# B&R Automation Studio project AS_Target_Simulink_Test (part 5)

#### TD_Test.c
```c
/********************************************************************
 * COPYRIGHT -- Bernecker + Rainer Industrie-Elektronik Ges.m.b.H.
 ********************************************************************
 * Program: TransmissionDownshiftTestSequence
 * File: TD_Test.c
 * Author: The MathWorks, Inc.
 * Created: Wed Jun 03 01:12:01 1998
 ********************************************************************
 * Implementation of program TransmissionDownshiftTestSequence
 ********************************************************************
 * Generated with B&R Automation Studio Target for Simulink  V6.1.0
 * (ERT based)
 ********************************************************************/

#define _ASMATH_
#define ASMATH_
#define _ASMATH_H
#define ASMATH_H
#define _ASMATH_H_
#define ASMATH_H_
#define _ASSTRING_
#define ASSTRING_
#define _ASSTRING_H
#define ASSTRING_H
#define _ASSTRING_H_
#define ASSTRING_H_
#include <bur/plctypes.h>
#ifdef _DEFAULT_INCLUDES
#include <AsDefault.h>
#endif

#include "TransmissionDownshiftTestSequence.h"
#include "rtwtypes.h"

/*  Defines */

/*  Data Types */

/**************************** GLOBAL DATA *************************************/
/*  Definitions */

/*  Declarations  */

/***************************** FILE SCOPE DATA ********************************/

/*************************** FUNCTIONS ****************************************/
#ifdef __cplusplus

unsigned long bur_heap_size = 6553500;

#endif

  void _INIT mainINIT(void)
{

    UDINT st_ident;
  RTInfo_typ rt_info;
  rt_info.enable = 1;
  RTInfo(&rt_info);
  if (rt_info.cycle_time != 10000) {
    /* cycle time does not match Simulink fixed-step size */
    ST_ident("TD_Test", 0, &st_ident);
    ST_tmp_suspend(st_ident);
    ERR_warning(33310, 0);
  }

  /* initialize model */
  TransmissionDownshiftTestSequence_initialize();

} void _CYCLIC mainCYCLIC(void)
{
  /* call model step function */
  TransmissionDownshiftTestSequence_output();

  TransmissionDownshiftTestSequence_update();

} void _EXIT mainEXIT(void)
{
  /* terminate model */
  TransmissionDownshiftTestSequence_terminate();

} /*****************************************************************************
     Task sample time: 0.01s
   *****************************************************************************/
/*****************************************************************************
   B&R Automation Studio Target for Simulink Version: V6.1.0 (06-Nov-2019)
 *****************************************************************************/

/*======================== TOOL VERSION INFORMATION ==========================*
 * MATLAB 9.7 (R2019b)18-Jul-2019                                             *
 * Simulink 10.0 (R2019b)18-Jul-2019                                          *
 * Simulink Coder 9.2 (R2019b)18-Jul-2019                                     *
 * Embedded Coder 7.3 (R2019b)18-Jul-2019                                     *
 * Stateflow 10.1 (R2019b)18-Jul-2019                                         *
 * Fixed-Point Designer 6.4 (R2019b)18-Jul-2019                               *
 *============================================================================*/

/*======================= LICENSE IN USE INFORMATION =========================*
 * matlab                                                                     *
 * matlab_coder                                                               *
 * real-time_workshop                                                         *
 * rtw_embedded_coder                                                         *
 * simulink                                                                   *
 * simulink_test                                                              *
 * stateflow                                                                  *
 *============================================================================*/
```

#### TransmissionDownshiftTestSequence.c
```c
/********************************************************************
 * COPYRIGHT -- Bernecker + Rainer Industrie-Elektronik Ges.m.b.H.
 ********************************************************************
 * Program: TransmissionDownshiftTestSequence
 * File: TransmissionDownshiftTestSequence.c
 * Author: The MathWorks, Inc.
 * Created: Wed Jun 03 01:12:01 1998
 ********************************************************************
 * Implementation of program TransmissionDownshiftTestSequence
 ********************************************************************
 * Generated with B&R Automation Studio Target for Simulink  V6.1.0
 * (ERT based)
 ********************************************************************/

#include "TransmissionDownshiftTestSequence.h"
#include "TransmissionDownshiftTestSequence_private.h"

/*  Defines */

/* Named constants for Chart: '<Root>/shift_controller' */
#define TransmissionDow_IN_downshifting ((uint8_T)1U)
#define TransmissionDow_IN_steady_state ((uint8_T)2U)
#define TransmissionDowns_IN_upshifting ((uint8_T)3U)
#define TransmissionDownshif_event_DOWN (0)
#define TransmissionDownshiftT_event_UP (1)
#define Transmission_IN_NO_ACTIVE_CHILD ((uint8_T)0U)

/*  Data Types */

/**************************** GLOBAL DATA *************************************/
/*  Definitions */

/* Block signals (default storage) */
BlockIO_TransmissionDownshiftTe TransmissionDownshiftTestSequ_B;

/* Continuous states */
ContinuousStates_TransmissionDo TransmissionDownshiftTestSequ_X;

/* Block states (default storage) */
D_Work_TransmissionDownshiftTes TransmissionDownshiftTest_DWork;

/* External inputs (root inport signals with default storage) */
ExternalInputs_TransmissionDown TransmissionDownshiftTestSequ_U;

/* External outputs (root outports fed by signals with default storage) */
ExternalOutputs_TransmissionDow TransmissionDownshiftTestSequ_Y;

/* Real-time model */
RT_MODEL_TransmissionDownshiftT TransmissionDownshiftTestSeq_M_;
RT_MODEL_TransmissionDownshiftT *const TransmissionDownshiftTestSeq_M =
  &TransmissionDownshiftTestSeq_M_;

/*  Declarations  */

/* Forward declaration for local functions */
static void TransmissionDownshif_gear_state(const int32_T *sfEvent);
static void rate_scheduler(void);

/***************************** FILE SCOPE DATA ********************************/

/*************************** FUNCTIONS ****************************************/
real_T look1_binlxpw(real_T u0, const real_T bp0[], const real_T table[],
                     uint32_T maxIndex)
{
  real_T frac;
  uint32_T iRght;
  uint32_T iLeft;
  uint32_T bpIdx;

  /* Column-major Lookup 1-D
     Search method: 'binary'
     Use previous index: 'off'
     Interpolation method: 'Linear point-slope'
     Extrapolation method: 'Linear'
     Use last breakpoint for index at or above upper limit: 'off'
     Remove protection against out-of-range input in generated code: 'off'
   */
  /* Prelookup - Index and Fraction
     Index Search method: 'binary'
     Extrapolation method: 'Linear'
     Use previous index: 'off'
     Use last breakpoint for index at or above upper limit: 'off'
     Remove protection against out-of-range input in generated code: 'off'
   */
  if (u0 <= bp0[0U]) {
    iLeft = 0U;
    frac = (u0 - bp0[0U]) / (bp0[1U] - bp0[0U]);
  } else if (u0 < bp0[maxIndex]) {
    /* Binary Search */
    bpIdx = maxIndex >> 1U;
    iLeft = 0U;
    iRght = maxIndex;
    while (iRght - iLeft > 1U) {
      if (u0 < bp0[bpIdx]) {
        iRght = bpIdx;
      } else {
        iLeft = bpIdx;
      }

      bpIdx = (iRght + iLeft) >> 1U;
    }

    frac = (u0 - bp0[iLeft]) / (bp0[iLeft + 1U] - bp0[iLeft]);
  } else {
    iLeft = maxIndex - 1U;
    frac = (u0 - bp0[maxIndex - 1U]) / (bp0[maxIndex] - bp0[maxIndex - 1U]);
  }

  /* Column-major Interpolation 1-D
     Interpolation method: 'Linear point-slope'
     Use last breakpoint for index at or above upper limit: 'off'
     Overflow mode: 'portable wrapping'
   */
  return (table[iLeft + 1U] - table[iLeft]) * frac + table[iLeft];
}

real_T look2_binlxpw(real_T u0, real_T u1, const real_T bp0[], const real_T bp1[],
                     const real_T table[], const uint32_T maxIndex[], uint32_T
                     stride)
{
  real_T frac;
  uint32_T bpIndices[2];
  real_T fractions[2];
  real_T yL_1d;
  uint32_T iRght;
  uint32_T bpIdx;
  uint32_T iLeft;

  /* Column-major Lookup 2-D
     Search method: 'binary'
     Use previous index: 'off'
     Interpolation method: 'Linear point-slope'
     Extrapolation method: 'Linear'
     Use last breakpoint for index at or above upper limit: 'off'
     Remove protection against out-of-range input in generated code: 'off'
   */
  /* Prelookup - Index and Fraction
     Index Search method: 'binary'
     Extrapolation method: 'Linear'
     Use previous index: 'off'
     Use last breakpoint for index at or above upper limit: 'off'
     Remove protection against out-of-range input in generated code: 'off'
   */
  if (u0 <= bp0[0U]) {
    iLeft = 0U;
    frac = (u0 - bp0[0U]) / (bp0[1U] - bp0[0U]);
  } else if (u0 < bp0[maxIndex[0U]]) {
    /* Binary Search */
    bpIdx = maxIndex[0U] >> 1U;
    iLeft = 0U;
    iRght = maxIndex[0U];
    while (iRght - iLeft > 1U) {
      if (u0 < bp0[bpIdx]) {
        iRght = bpIdx;
      } else {
        iLeft = bpIdx;
      }

      bpIdx = (iRght + iLeft) >> 1U;
    }

    frac = (u0 - bp0[iLeft]) / (bp0[iLeft + 1U] - bp0[iLeft]);
  } else {
    iLeft = maxIndex[0U] - 1U;
    frac = (u0 - bp0[maxIndex[0U] - 1U]) / (bp0[maxIndex[0U]] - bp0[maxIndex[0U]
      - 1U]);
  }

  fractions[0U] = frac;
  bpIndices[0U] = iLeft;

  /* Prelookup - Index and Fraction
     Index Search method: 'binary'
     Extrapolation method: 'Linear'
     Use previous index: 'off'
     Use last breakpoint for index at or above upper limit: 'off'
     Remove protection against out-of-range input in generated code: 'off'
   */
  if (u1 <= bp1[0U]) {
    iLeft = 0U;
    frac = (u1 - bp1[0U]) / (bp1[1U] - bp1[0U]);
  } else if (u1 < bp1[maxIndex[1U]]) {
    /* Binary Search */
    bpIdx = maxIndex[1U] >> 1U;
    iLeft = 0U;
    iRght = maxIndex[1U];
    while (iRght - iLeft > 1U) {
      if (u1 < bp1[bpIdx]) {
        iRght = bpIdx;
      } else {
        iLeft = bpIdx;
      }

      bpIdx = (iRght + iLeft) >> 1U;
    }

    frac = (u1 - bp1[iLeft]) / (bp1[iLeft + 1U] - bp1[iLeft]);
  } else {
    iLeft = maxIndex[1U] - 1U;
    frac = (u1 - bp1[maxIndex[1U] - 1U]) / (bp1[maxIndex[1U]] - bp1[maxIndex[1U]
      - 1U]);
  }

  /* Column-major Interpolation 2-D
     Interpolation method: 'Linear point-slope'
     Use last breakpoint for index at or above upper limit: 'off'
     Overflow mode: 'portable wrapping'
   */
  bpIdx = iLeft * stride + bpIndices[0U];
  yL_1d = (table[bpIdx + 1U] - table[bpIdx]) * fractions[0U] + table[bpIdx];
  bpIdx += stride;
  return (((table[bpIdx + 1U] - table[bpIdx]) * fractions[0U] + table[bpIdx]) -
          yL_1d) * frac + yL_1d;
}

/*
 *   This function updates active task flag for each subrate.
 * The function is called at model base rate, hence the
 * generated code self-manages all its subrates.
 */
static void rate_scheduler(void)
{
  /* Compute which subrates run during the next base time step.  Subrates
   * are an integer multiple of the base rate counter.  Therefore, the subtask
   * counter is reset when it reaches its limit (zero means run).
   */
  (TransmissionDownshiftTestSeq_M->Timing.TaskCounters.TID[2])++;
  if ((TransmissionDownshiftTestSeq_M->Timing.TaskCounters.TID[2]) > 3) {/* Sample time: [0.04s, 0.0s] */
    TransmissionDownshiftTestSeq_M->Timing.TaskCounters.TID[2] = 0;
  }
}

/*
 * This function updates continuous states using the ODE1 fixed-step
 * solver algorithm
 */
static void rt_ertODEUpdateContinuousStates(RTWSolverInfo *si )
{
  time_T tnew = rtsiGetSolverStopTime(si);
  time_T h = rtsiGetStepSize(si);
  real_T *x = rtsiGetContStates(si);
  ODE1_IntgData *id = (ODE1_IntgData *)rtsiGetSolverData(si);
  real_T *f0 = id->f[0];
  int_T i;
  int_T nXc = 2;
  rtsiSetSimTimeStep(si,MINOR_TIME_STEP);
  rtsiSetdX(si, f0);
  TransmissionDownshiftTestSequence_derivatives();
  rtsiSetT(si, tnew);
  for (i = 0; i < nXc; ++i) {
    x[i] += h * f0[i];
  }

  rtsiSetSimTimeStep(si,MAJOR_TIME_STEP);
}

/* Function for Chart: '<Root>/shift_controller' */
static void TransmissionDownshif_gear_state(const int32_T *sfEvent)
{
  switch (TransmissionDownshiftTestSequ_B.gear) {
   case gearType_first:
    if (*sfEvent == TransmissionDownshiftT_event_UP) {
      TransmissionDownshiftTestSequ_B.gear = gearType_second;
    }
    break;

   case gearType_second:
    if (*sfEvent == TransmissionDownshiftT_event_UP) {
      TransmissionDownshiftTestSequ_B.gear = gearType_third;
    } else {
      if (*sfEvent == TransmissionDownshif_event_DOWN) {
        TransmissionDownshiftTestSequ_B.gear = gearType_first;
      }
    }
    break;

   case gearType_third:
    if (*sfEvent == TransmissionDownshiftT_event_UP) {
      TransmissionDownshiftTestSequ_B.gear = gearType_fourth;
    } else {
      if (*sfEvent == TransmissionDownshif_event_DOWN) {
        TransmissionDownshiftTestSequ_B.gear = gearType_second;
      }
    }
    break;

   case gearType_fourth:
    if (*sfEvent == TransmissionDownshif_event_DOWN) {
      TransmissionDownshiftTestSequ_B.gear = gearType_third;
    }
    break;

   default:
    /* Unreachable state, for coverage only */
    TransmissionDownshiftTestSequ_B.gear = gearType_None;
    break;
  }
}

/* Model output function */
void TransmissionDownshiftTestSequence_output(void)
{
  real_T rtb_out;
  real_T mph;
  int32_T sfEvent;
  real_T interp_down;
  real_T mph_0;
  if (rtmIsMajorTimeStep(TransmissionDownshiftTestSeq_M)) {
    /* set solver stop time */
    if (!(TransmissionDownshiftTestSeq_M->Timing.clockTick0+1)) {
      rtsiSetSolverStopTime(&TransmissionDownshiftTestSeq_M->solverInfo,
                            ((TransmissionDownshiftTestSeq_M->Timing.clockTickH0
        + 1) * TransmissionDownshiftTestSeq_M->Timing.stepSize0 * 4294967296.0));
    } else {
      rtsiSetSolverStopTime(&TransmissionDownshiftTestSeq_M->solverInfo,
                            ((TransmissionDownshiftTestSeq_M->Timing.clockTick0
        + 1) * TransmissionDownshiftTestSeq_M->Timing.stepSize0 +
        TransmissionDownshiftTestSeq_M->Timing.clockTickH0 *
        TransmissionDownshiftTestSeq_M->Timing.stepSize0 * 4294967296.0));
    }
  }                                    /* end MajorTimeStep */

  /* Update absolute time of base rate at minor time step */
  if (rtmIsMinorTimeStep(TransmissionDownshiftTestSeq_M)) {
    TransmissionDownshiftTestSeq_M->Timing.t[0] = rtsiGetT
      (&TransmissionDownshiftTestSeq_M->solverInfo);
  }

  /* Gain: '<S6>/mph' incorporates:
   *  Gain: '<S6>/linear speed'
   *  Integrator: '<S6>/wheel speed'
   */
  mph = 6.2831853071795862 * TransmissionDownshiftTestSequ_P.vehicledata[3] *
    TransmissionDownshiftTestSequ_X.wheelspeed_CSTATE *
    TransmissionDownshiftTestSequ_P.mph_Gain;

  /* Outport: '<Root>/Out1' */
  TransmissionDownshiftTestSequ_Y.Out1 = mph;
  if (rtmIsMajorTimeStep(TransmissionDownshiftTestSeq_M) &&
      TransmissionDownshiftTestSeq_M->Timing.TaskCounters.TID[2] == 0) {
    /* Chart: '<Root>/shift_controller' */
    sfEvent = -1;
    if (TransmissionDownshiftTest_DWork.temporalCounter_i1 < 255U) {
      TransmissionDownshiftTest_DWork.temporalCounter_i1++;
    }

    if (TransmissionDownshiftTest_DWork.is_active_c4_TransmissionDownsh == 0U) {
      TransmissionDownshiftTest_DWork.is_active_c4_TransmissionDownsh = 1U;
      TransmissionDownshiftTest_DWork.is_active_gear_state = 1U;
      TransmissionDownshiftTestSequ_B.gear = gearType_first;
      TransmissionDownshiftTest_DWork.is_active_selection_state = 1U;
      TransmissionDownshiftTest_DWork.is_selection_state =
        TransmissionDow_IN_steady_state;
    } else {
      if (TransmissionDownshiftTest_DWork.is_active_gear_state != 0U) {
        TransmissionDownshif_gear_state(&sfEvent);
      }

      if (TransmissionDownshiftTest_DWork.is_active_selection_state != 0U) {
        /* Outputs for Function Call SubSystem: '<S1>/selection_state.calc_th' */
        /* MATLAB Function: '<S3>/Look-Up' */
        switch (TransmissionDownshiftTestSequ_B.gear) {
         case gearType_fourth:
          rtb_out = 4.0;
          break;

         case gearType_third:
          rtb_out = 3.0;
          break;

         case gearType_second:
          rtb_out = 2.0;
          break;

         default:
          rtb_out = 1.0;
          break;
        }

        /* End of MATLAB Function: '<S3>/Look-Up' */

        /* Lookup_n-D: '<S3>/interp_down' incorporates:
         *  Inport: '<Root>/throttle'
         */
        interp_down = look2_binlxpw(TransmissionDownshiftTestSequ_U.throttle,
          rtb_out, TransmissionDownshiftTestSequ_P.downth,
          TransmissionDownshiftTestSequ_P.interp_down_bp02Data,
          TransmissionDownshiftTestSequ_P.downtab,
          TransmissionDownshiftTestSequ_P.interp_down_maxIndex, 6U);

        /* Lookup_n-D: '<S3>/interp_up' incorporates:
         *  Inport: '<Root>/throttle'
         */
        rtb_out = look2_binlxpw(TransmissionDownshiftTestSequ_U.throttle,
          rtb_out, TransmissionDownshiftTestSequ_P.upth,
          TransmissionDownshiftTestSequ_P.interp_up_bp02Data,
          TransmissionDownshiftTestSequ_P.uptab,
          TransmissionDownshiftTestSequ_P.interp_up_maxIndex, 6U);

        /* End of Outputs for SubSystem: '<S1>/selection_state.calc_th' */
        switch (TransmissionDownshiftTest_DWork.is_selection_state) {
         case TransmissionDow_IN_downshifting:
          if ((TransmissionDownshiftTest_DWork.temporalCounter_i1 >=
               TransmissionDownshiftTestSequ_P.shift_controller_TWAIT) && (mph <=
               interp_down)) {
            sfEvent = TransmissionDownshif_event_DOWN;
            if (TransmissionDownshiftTest_DWork.is_active_gear_state != 0U) {
              TransmissionDownshif_gear_state(&sfEvent);
            }

            TransmissionDownshiftTest_DWork.is_selection_state =
              TransmissionDow_IN_steady_state;
          } else {
            if (mph > interp_down) {
              TransmissionDownshiftTest_DWork.is_selection_state =
                TransmissionDow_IN_steady_state;
            }
          }
          break;

         case TransmissionDow_IN_steady_state:
          if (mph > rtb_out) {
            TransmissionDownshiftTest_DWork.is_selection_state =
              TransmissionDowns_IN_upshifting;
            TransmissionDownshiftTest_DWork.temporalCounter_i1 = 0U;
          } else {
            if (mph < interp_down) {
              TransmissionDownshiftTest_DWork.is_selection_state =
                TransmissionDow_IN_downshifting;
              TransmissionDownshiftTest_DWork.temporalCounter_i1 = 0U;
            }
          }
          break;

         case TransmissionDowns_IN_upshifting:
          if ((TransmissionDownshiftTest_DWork.temporalCounter_i1 >=
               TransmissionDownshiftTestSequ_P.shift_controller_TWAIT) && (mph >=
               rtb_out)) {
            sfEvent = TransmissionDownshiftT_event_UP;
            if (TransmissionDownshiftTest_DWork.is_active_gear_state != 0U) {
              TransmissionDownshif_gear_state(&sfEvent);
            }

            TransmissionDownshiftTest_DWork.is_selection_state =
              TransmissionDow_IN_steady_state;
          } else {
            if (mph < rtb_out) {
              TransmissionDownshiftTest_DWork.is_selection_state =
                TransmissionDow_IN_steady_state;
            }
          }
          break;

         default:
          /* Unreachable state, for coverage only */
          TransmissionDownshiftTest_DWork.is_selection_state =
            Transmission_IN_NO_ACTIVE_CHILD;
          break;
        }
      }
    }

    /* End of Chart: '<Root>/shift_controller' */

    /* MATLAB Function: '<S9>/Look-Up Table' */
    switch (TransmissionDownshiftTestSequ_B.gear) {
     case gearType_fourth:
      TransmissionDownshiftTestSequ_B.out = 0.677;
      break;

     case gearType_third:
      TransmissionDownshiftTestSequ_B.out = 1.0;
      break;

     case gearType_second:
      TransmissionDownshiftTestSequ_B.out = 1.45;
      break;

     default:
      TransmissionDownshiftTestSequ_B.out = 2.393;
      break;
    }

    /* End of MATLAB Function: '<S9>/Look-Up Table' */
  }

  /* Integrator: '<S5>/Integrator' */
  /* Limited  Integrator  */
  if (TransmissionDownshiftTestSequ_X.Integrator_CSTATE >=
      TransmissionDownshiftTestSequ_P.Integrator_UpperSat) {
    TransmissionDownshiftTestSequ_X.Integrator_CSTATE =
      TransmissionDownshiftTestSequ_P.Integrator_UpperSat;
  } else {
    if (TransmissionDownshiftTestSequ_X.Integrator_CSTATE <=
        TransmissionDownshiftTestSequ_P.Integrator_LowerSat) {
      TransmissionDownshiftTestSequ_X.Integrator_CSTATE =
        TransmissionDownshiftTestSequ_P.Integrator_LowerSat;
    }
  }

  /* Product: '<S8>/speed ratio' incorporates:
   *  Gain: '<S6>/final drive ratio2'
   *  Integrator: '<S5>/Integrator'
   *  Integrator: '<S6>/wheel speed'
   *  Product: '<S9>/Product1'
   */
  interp_down = TransmissionDownshiftTestSequ_P.vehicledata[0] *
    TransmissionDownshiftTestSequ_X.wheelspeed_CSTATE *
    TransmissionDownshiftTestSequ_B.out /
    TransmissionDownshiftTestSequ_X.Integrator_CSTATE;

  /* Fcn: '<S8>/impeller' incorporates:
   *  Integrator: '<S5>/Integrator'
   *  Lookup_n-D: '<S8>/K factor'
   *  Product: '<S8>/quotient'
   */
  rtb_out = pow(TransmissionDownshiftTestSequ_X.Integrator_CSTATE /
                look1_binlxpw(interp_down,
    TransmissionDownshiftTestSequ_P.TorqueConverter_speedratio,
    TransmissionDownshiftTestSequ_P.TorqueConverter_Kfactor, 20U), 2.0);

  /* Gain: '<S5>/engine + impeller inertia' incorporates:
   *  Fcn: '<S8>/impeller'
   *  Inport: '<Root>/throttle'
   *  Integrator: '<S5>/Integrator'
   *  Lookup_n-D: '<S5>/engine torque'
   *  Sum: '<S5>/Sum'
   */
  TransmissionDownshiftTestSequ_B.engineimpellerinertia = 1.0 /
    TransmissionDownshiftTestSequ_P.Iei * (look2_binlxpw
    (TransmissionDownshiftTestSequ_U.throttle,
     TransmissionDownshiftTestSequ_X.Integrator_CSTATE,
     TransmissionDownshiftTestSequ_P.thvec,
     TransmissionDownshiftTestSequ_P.nevec, TransmissionDownshiftTestSequ_P.emap,
     TransmissionDownshiftTestSequ_P.enginetorque_maxIndex, 10U) - rtb_out);

  /* Lookup_n-D: '<S8>/Torque ratio' */
  interp_down = look1_binlxpw(interp_down,
    TransmissionDownshiftTestSequ_P.TorqueConverter_speedratio,
    TransmissionDownshiftTestSequ_P.TorqueConverter_Torkratio, 20U);

  /* Signum: '<S6>/Sign' */
  if (mph < 0.0) {
    mph_0 = -1.0;
  } else if (mph > 0.0) {
    mph_0 = 1.0;
  } else {
    mph_0 = mph;
  }

  /* End of Signum: '<S6>/Sign' */

  /* Gain: '<S6>/vehicle inertia' incorporates:
   *  Fcn: '<S6>/road load'
   *  Fcn: '<S8>/impeller'
   *  Gain: '<S6>/final drive ratio1'
   *  Inport: '<Root>/brake'
   *  Product: '<S6>/signed load'
   *  Product: '<S8>/turbine'
   *  Product: '<S9>/Product'
   *  Sum: '<S6>/Sum'
   *  Sum: '<S6>/Sum1'
   */
  TransmissionDownshiftTestSequ_B.vehicleinertia = (rtb_out * interp_down *
    TransmissionDownshiftTestSequ_B.out *
    TransmissionDownshiftTestSequ_P.vehicledata[0] - ((0.3 * pow(mph, 2.0) +
    40.0) + TransmissionDownshiftTestSequ_U.brake) * mph_0) * (1.0 /
    TransmissionDownshiftTestSequ_P.vehicledata[4]);
  if (rtmIsMajorTimeStep(TransmissionDownshiftTestSeq_M) &&
      TransmissionDownshiftTestSeq_M->Timing.TaskCounters.TID[1] == 0) {
  }

  /* Outport: '<Root>/Out2' incorporates:
   *  Inport: '<Root>/throttle'
   */
  TransmissionDownshiftTestSequ_Y.Out2 =
    TransmissionDownshiftTestSequ_U.throttle;
}

/* Model update function */
void TransmissionDownshiftTestSequence_update(void)
{
  if (rtmIsMajorTimeStep(TransmissionDownshiftTestSeq_M)) {
    rt_ertODEUpdateContinuousStates(&TransmissionDownshiftTestSeq_M->solverInfo);
  }

  /* Update absolute time for base rate */
  /* The "clockTick0" counts the number of times the code of this task has
   * been executed. The absolute time is the multiplication of "clockTick0"
   * and "Timing.stepSize0". Size of "clockTick0" ensures timer will not
   * overflow during the application lifespan selected.
   * Timer of this task consists of two 32 bit unsigned integers.
   * The two integers represent the low bits Timing.clockTick0 and the high bits
   * Timing.clockTickH0. When the low bit overflows to 0, the high bits increment.
   */
  if (!(++TransmissionDownshiftTestSeq_M->Timing.clockTick0)) {
    ++TransmissionDownshiftTestSeq_M->Timing.clockTickH0;
  }

  TransmissionDownshiftTestSeq_M->Timing.t[0] = rtsiGetSolverStopTime
    (&TransmissionDownshiftTestSeq_M->solverInfo);

  {
    /* Update absolute timer for sample time: [0.01s, 0.0s] */
    /* The "clockTick1" counts the number of times the code of this task has
     * been executed. The resolution of this integer timer is 0.01, which is the step size
     * of the task. Size of "clockTick1" ensures timer will not overflow during the
     * application lifespan selected.
     * Timer of this task consists of two 32 bit unsigned integers.
     * The two integers represent the low bits Timing.clockTick1 and the high bits
     * Timing.clockTickH1. When the low bit overflows to 0, the high bits increment.
     */
    TransmissionDownshiftTestSeq_M->Timing.clockTick1++;
    if (!TransmissionDownshiftTestSeq_M->Timing.clockTick1) {
      TransmissionDownshiftTestSeq_M->Timing.clockTickH1++;
    }
  }

  rate_scheduler();
}

/* Derivatives for root system: '<Root>' */
void TransmissionDownshiftTestSequence_derivatives(void)
{
  boolean_T lsat;
  boolean_T usat;
  StateDerivatives_TransmissionDo *_rtXdot;
  _rtXdot = ((StateDerivatives_TransmissionDo *)
             TransmissionDownshiftTestSeq_M->derivs);

  /* Derivatives for Integrator: '<S6>/wheel speed' */
  _rtXdot->wheelspeed_CSTATE = TransmissionDownshiftTestSequ_B.vehicleinertia;

  /* Derivatives for Integrator: '<S5>/Integrator' */
  lsat = (TransmissionDownshiftTestSequ_X.Integrator_CSTATE <=
          TransmissionDownshiftTestSequ_P.Integrator_LowerSat);
  usat = (TransmissionDownshiftTestSequ_X.Integrator_CSTATE >=
          TransmissionDownshiftTestSequ_P.Integrator_UpperSat);
  if (((!lsat) && (!usat)) || (lsat &&
       (TransmissionDownshiftTestSequ_B.engineimpellerinertia > 0.0)) || (usat &&
       (TransmissionDownshiftTestSequ_B.engineimpellerinertia < 0.0))) {
    _rtXdot->Integrator_CSTATE =
      TransmissionDownshiftTestSequ_B.engineimpellerinertia;
  } else {
    /* in saturation */
    _rtXdot->Integrator_CSTATE = 0.0;
  }

  /* End of Derivatives for Integrator: '<S5>/Integrator' */
}

/* Model initialize function */
void TransmissionDownshiftTestSequence_initialize(void)
{
  /* Registration code */
  {
    /* Setup solver object */
    rtsiSetSimTimeStepPtr(&TransmissionDownshiftTestSeq_M->solverInfo,
                          &TransmissionDownshiftTestSeq_M->Timing.simTimeStep);
    rtsiSetTPtr(&TransmissionDownshiftTestSeq_M->solverInfo, &rtmGetTPtr
                (TransmissionDownshiftTestSeq_M));
    rtsiSetStepSizePtr(&TransmissionDownshiftTestSeq_M->solverInfo,
                       &TransmissionDownshiftTestSeq_M->Timing.stepSize0);
    rtsiSetdXPtr(&TransmissionDownshiftTestSeq_M->solverInfo,
                 &TransmissionDownshiftTestSeq_M->derivs);
    rtsiSetContStatesPtr(&TransmissionDownshiftTestSeq_M->solverInfo, (real_T **)
                         &TransmissionDownshiftTestSeq_M->contStates);
    rtsiSetNumContStatesPtr(&TransmissionDownshiftTestSeq_M->solverInfo,
      &TransmissionDownshiftTestSeq_M->Sizes.numContStates);
    rtsiSetNumPeriodicContStatesPtr(&TransmissionDownshiftTestSeq_M->solverInfo,
      &TransmissionDownshiftTestSeq_M->Sizes.numPeriodicContStates);
    rtsiSetPeriodicContStateIndicesPtr
      (&TransmissionDownshiftTestSeq_M->solverInfo,
       &TransmissionDownshiftTestSeq_M->periodicContStateIndices);
    rtsiSetPeriodicContStateRangesPtr
      (&TransmissionDownshiftTestSeq_M->solverInfo,
       &TransmissionDownshiftTestSeq_M->periodicContStateRanges);
    rtsiSetErrorStatusPtr(&TransmissionDownshiftTestSeq_M->solverInfo,
                          (&rtmGetErrorStatus(TransmissionDownshiftTestSeq_M)));
    rtsiSetRTModelPtr(&TransmissionDownshiftTestSeq_M->solverInfo,
                      TransmissionDownshiftTestSeq_M);
  }

  rtsiSetSimTimeStep(&TransmissionDownshiftTestSeq_M->solverInfo,
                     MAJOR_TIME_STEP);
  TransmissionDownshiftTestSeq_M->intgData.f[0] =
    TransmissionDownshiftTestSeq_M->odeF[0];
  TransmissionDownshiftTestSeq_M->contStates = ((ContinuousStates_TransmissionDo
    *) &TransmissionDownshiftTestSequ_X);
  rtsiSetSolverData(&TransmissionDownshiftTestSeq_M->solverInfo, (void *)
                    &TransmissionDownshiftTestSeq_M->intgData);
  rtsiSetSolverName(&TransmissionDownshiftTestSeq_M->solverInfo,"ode1");
  rtmSetTPtr(TransmissionDownshiftTestSeq_M,
             &TransmissionDownshiftTestSeq_M->Timing.tArray[0]);
  TransmissionDownshiftTestSeq_M->Timing.stepSize0 = 0.01;

  /* InitializeConditions for Integrator: '<S6>/wheel speed' */
  TransmissionDownshiftTestSequ_X.wheelspeed_CSTATE =
    TransmissionDownshiftTestSequ_P.vehicledata[5] /
    TransmissionDownshiftTestSequ_P.vehicledata[3] *
    TransmissionDownshiftTestSequ_P.vehicledata[0] /
    TransmissionDownshiftTestSequ_P.vehicledata[0];

  /* InitializeConditions for Integrator: '<S5>/Integrator' */
  TransmissionDownshiftTestSequ_X.Integrator_CSTATE =
    TransmissionDownshiftTestSequ_P.Integrator_IC;

  /* SystemInitialize for Chart: '<Root>/shift_controller' */
  TransmissionDownshiftTestSequ_B.gear = gearType_None;
}

/* Model terminate function */
void TransmissionDownshiftTestSequence_terminate(void)
{
  /* (no terminate code required) */
}

/*======================== TOOL VERSION INFORMATION ==========================*
 * MATLAB 9.7 (R2019b)18-Jul-2019                                             *
 * Simulink 10.0 (R2019b)18-Jul-2019                                          *
 * Simulink Coder 9.2 (R2019b)18-Jul-2019                                     *
 * Embedded Coder 7.3 (R2019b)18-Jul-2019                                     *
 * Stateflow 10.1 (R2019b)18-Jul-2019                                         *
 * Fixed-Point Designer 6.4 (R2019b)18-Jul-2019                               *
 *============================================================================*/

/*======================= LICENSE IN USE INFORMATION =========================*
 * matlab                                                                     *
 * matlab_coder                                                               *
 * real-time_workshop                                                         *
 * rtw_embedded_coder                                                         *
 * simulink                                                                   *
 * simulink_test                                                              *
 * stateflow                                                                  *
 *============================================================================*/
```

#### TransmissionDownshiftTestSequence.h
```c
/********************************************************************
 * COPYRIGHT -- Bernecker + Rainer Industrie-Elektronik Ges.m.b.H.
 ********************************************************************
 * Program: TransmissionDownshiftTestSequence
 * File: TransmissionDownshiftTestSequence.h
 * Author: The MathWorks, Inc.
 * Created: Wed Jun 03 01:12:01 1998
 ********************************************************************
 * Header for program TransmissionDownshiftTestSequence
 ********************************************************************
 * Generated with B&R Automation Studio Target for Simulink  V6.1.0
 * (ERT based)
 ********************************************************************/

#ifndef RTW_HEADER_TransmissionDownshiftTestSequence_h_
#define RTW_HEADER_TransmissionDownshiftTestSequence_h_
#include <math.h>
#ifndef TransmissionDownshiftTestSequence_COMMON_INCLUDES_
# define TransmissionDownshiftTestSequence_COMMON_INCLUDES_
#include "rtwtypes.h"
#include "rtw_continuous.h"
#include "rtw_solver.h"
#endif                  /* TransmissionDownshiftTestSequence_COMMON_INCLUDES_ */

#include <bur/plctypes.h>

#ifdef _DEFAULT_INCLUDES
 #include <AsDefault.h>
#endif

#ifndef AST_ROUND
#define AST_ROUND(x) ((x)>=0?(long long)((x)+0.5):(long long)((x)-0.5))
#endif

#include "TransmissionDownshiftTestSequence_types.h"

/* Macros for accessing real-time model data structure */
#ifndef rtmGetContStateDisabled
# define rtmGetContStateDisabled(rtm)  ((rtm)->contStateDisabled)
#endif

#ifndef rtmSetContStateDisabled
# define rtmSetContStateDisabled(rtm, val) ((rtm)->contStateDisabled = (val))
#endif

#ifndef rtmGetContStates
# define rtmGetContStates(rtm)         ((rtm)->contStates)
#endif

#ifndef rtmSetContStates
# define rtmSetContStates(rtm, val)    ((rtm)->contStates = (val))
#endif

#ifndef rtmGetContTimeOutputInconsistentWithStateAtMajorStepFlag
# define rtmGetContTimeOutputInconsistentWithStateAtMajorStepFlag(rtm) ((rtm)->CTOutputIncnstWithState)
#endif

#ifndef rtmSetContTimeOutputInconsistentWithStateAtMajorStepFlag
# define rtmSetContTimeOutputInconsistentWithStateAtMajorStepFlag(rtm, val) ((rtm)->CTOutputIncnstWithState = (val))
#endif

#ifndef rtmGetDerivCacheNeedsReset
# define rtmGetDerivCacheNeedsReset(rtm) ((rtm)->derivCacheNeedsReset)
#endif

#ifndef rtmSetDerivCacheNeedsReset
# define rtmSetDerivCacheNeedsReset(rtm, val) ((rtm)->derivCacheNeedsReset = (val))
#endif

#ifndef rtmGetIntgData
# define rtmGetIntgData(rtm)           ((rtm)->intgData)
#endif

#ifndef rtmSetIntgData
# define rtmSetIntgData(rtm, val)      ((rtm)->intgData = (val))
#endif

#ifndef rtmGetOdeF
# define rtmGetOdeF(rtm)               ((rtm)->odeF)
#endif

#ifndef rtmSetOdeF
# define rtmSetOdeF(rtm, val)          ((rtm)->odeF = (val))
#endif

#ifndef rtmGetPeriodicContStateIndices
# define rtmGetPeriodicContStateIndices(rtm) ((rtm)->periodicContStateIndices)
#endif

#ifndef rtmSetPeriodicContStateIndices
# define rtmSetPeriodicContStateIndices(rtm, val) ((rtm)->periodicContStateIndices = (val))
#endif

#ifndef rtmGetPeriodicContStateRanges
# define rtmGetPeriodicContStateRanges(rtm) ((rtm)->periodicContStateRanges)
#endif

#ifndef rtmSetPeriodicContStateRanges
# define rtmSetPeriodicContStateRanges(rtm, val) ((rtm)->periodicContStateRanges = (val))
#endif

#ifndef rtmGetZCCacheNeedsReset
# define rtmGetZCCacheNeedsReset(rtm)  ((rtm)->zCCacheNeedsReset)
#endif

#ifndef rtmSetZCCacheNeedsReset
# define rtmSetZCCacheNeedsReset(rtm, val) ((rtm)->zCCacheNeedsReset = (val))
#endif

#ifndef rtmGetdX
# define rtmGetdX(rtm)                 ((rtm)->derivs)
#endif

#ifndef rtmSetdX
# define rtmSetdX(rtm, val)            ((rtm)->derivs = (val))
#endif

#ifndef rtmGetErrorStatus
# define rtmGetErrorStatus(rtm)        ((rtm)->errorStatus)
#endif

#ifndef rtmSetErrorStatus
# define rtmSetErrorStatus(rtm, val)   ((rtm)->errorStatus = (val))
#endif

#ifndef rtmGetStopRequested
# define rtmGetStopRequested(rtm)      ((rtm)->Timing.stopRequestedFlag)
#endif

#ifndef rtmSetStopRequested
# define rtmSetStopRequested(rtm, val) ((rtm)->Timing.stopRequestedFlag = (val))
#endif

#ifndef rtmGetStopRequestedPtr
# define rtmGetStopRequestedPtr(rtm)   (&((rtm)->Timing.stopRequestedFlag))
#endif

#ifndef rtmGetT
# define rtmGetT(rtm)                  (rtmGetTPtr((rtm))[0])
#endif

#ifndef rtmGetTPtr
# define rtmGetTPtr(rtm)               ((rtm)->Timing.t)
#endif

#define TransmissionDownshiftTestSequence_M (TransmissionDownshiftTestSeq_M)
#ifndef MIN
#define MIN(a,b)                       ((a) < (b) ? (a) : (b))
#endif

#ifndef MAX
#define MAX(a,b)                       ((a) > (b) ? (a) : (b))
#endif

/* Block signals (default storage) */
typedef struct {
  real_T engineimpellerinertia;        /* '<S5>/engine + impeller inertia' */
  real_T vehicleinertia;               /* '<S6>/vehicle inertia' */
  real_T out;                          /* '<S9>/Look-Up Table' */
  gearType gear;                       /* '<Root>/shift_controller' */
} BlockIO_TransmissionDownshiftTe;

/* Block states (default storage) for system '<Root>' */
typedef struct {
  uint8_T is_active_c4_TransmissionDownsh;/* '<Root>/shift_controller' */
  uint8_T is_active_gear_state;        /* '<Root>/shift_controller' */
  uint8_T is_selection_state;          /* '<Root>/shift_controller' */
  uint8_T is_active_selection_state;   /* '<Root>/shift_controller' */
  uint8_T temporalCounter_i1;          /* '<Root>/shift_controller' */
} D_Work_TransmissionDownshiftTes;

/* Continuous states (default storage) */
typedef struct {
  real_T wheelspeed_CSTATE;            /* '<S6>/wheel speed' */
  real_T Integrator_CSTATE;            /* '<S5>/Integrator' */
} ContinuousStates_TransmissionDo;

/* State derivatives (default storage) */
typedef struct {
  real_T wheelspeed_CSTATE;            /* '<S6>/wheel speed' */
  real_T Integrator_CSTATE;            /* '<S5>/Integrator' */
} StateDerivatives_TransmissionDo;

/* State disabled  */
typedef struct {
  boolean_T wheelspeed_CSTATE;         /* '<S6>/wheel speed' */
  boolean_T Integrator_CSTATE;         /* '<S5>/Integrator' */
} StateDisabled_TransmissionDowns;

#ifndef ODE1_INTG
#define ODE1_INTG

/* ODE1 Integration Data */
typedef struct {
  real_T *f[1];                        /* derivatives */
} ODE1_IntgData;

#endif

/* External inputs (root inport signals with default storage) */
typedef struct {
  real_T brake;                        /* '<Root>/brake' */
  real_T throttle;                     /* '<Root>/throttle' */
} ExternalInputs_TransmissionDown;

/* External outputs (root outports fed by signals with default storage) */
typedef struct {
  real_T Out1;                         /* '<Root>/Out1' */
  real_T Out2;                         /* '<Root>/Out2' */
} ExternalOutputs_TransmissionDow;

/* Parameters (default storage) */
struct Parameters_TransmissionDownshif_ {
  real_T Iei;                          /* Variable: Iei
                                        * Referenced by: '<S5>/engine + impeller inertia'
                                        */
  real_T downtab[24];                  /* Variable: downtab
                                        * Referenced by: '<S3>/interp_down'
                                        */
  real_T downth[6];                    /* Variable: downth
                                        * Referenced by: '<S3>/interp_down'
                                        */
  real_T emap[110];                    /* Variable: emap
                                        * Referenced by: '<S5>/engine torque'
                                        */
  real_T nevec[11];                    /* Variable: nevec
                                        * Referenced by: '<S5>/engine torque'
                                        */
  real_T thvec[10];                    /* Variable: thvec
                                        * Referenced by: '<S5>/engine torque'
                                        */
  real_T uptab[24];                    /* Variable: uptab
                                        * Referenced by: '<S3>/interp_up'
                                        */
  real_T upth[6];                      /* Variable: upth
                                        * Referenced by: '<S3>/interp_up'
                                        */
  real_T vehicledata[6];               /* Variable: vehicledata
                                        * Referenced by:
                                        *   '<S6>/final drive ratio1'
                                        *   '<S6>/final drive ratio2'
                                        *   '<S6>/linear speed'
                                        *   '<S6>/vehicle inertia'
                                        *   '<S6>/wheel speed'
                                        */
  real_T TorqueConverter_Kfactor[21]; /* Mask Parameter: TorqueConverter_Kfactor
                                       * Referenced by: '<S8>/K factor'
                                       */
  real_T TorqueConverter_Torkratio[21];
                                    /* Mask Parameter: TorqueConverter_Torkratio
                                     * Referenced by: '<S8>/Torque ratio'
                                     */
  real_T TorqueConverter_speedratio[21];
                                   /* Mask Parameter: TorqueConverter_speedratio
                                    * Referenced by:
                                    *   '<S8>/K factor'
                                    *   '<S8>/Torque ratio'
                                    */
  uint8_T shift_controller_TWAIT;      /* Mask Parameter: shift_controller_TWAIT
                                        * Referenced by: '<Root>/shift_controller'
                                        */
  real_T interp_down_bp02Data[4];      /* Expression: [1:4]
                                        * Referenced by: '<S3>/interp_down'
                                        */
  real_T interp_up_bp02Data[4];        /* Expression: [1:4]
                                        * Referenced by: '<S3>/interp_up'
                                        */
  real_T mph_Gain;                     /* Expression: 60/5280
                                        * Referenced by: '<S6>/mph'
                                        */
  real_T Integrator_IC;                /* Expression: 1000
                                        * Referenced by: '<S5>/Integrator'
                                        */
  real_T Integrator_UpperSat;          /* Expression: 6000
                                        * Referenced by: '<S5>/Integrator'
                                        */
  real_T Integrator_LowerSat;          /* Expression: 600
                                        * Referenced by: '<S5>/Integrator'
                                        */
  uint32_T interp_down_maxIndex[2];  /* Computed Parameter: interp_down_maxIndex
                                      * Referenced by: '<S3>/interp_down'
                                      */
  uint32_T interp_up_maxIndex[2];      /* Computed Parameter: interp_up_maxIndex
                                        * Referenced by: '<S3>/interp_up'
                                        */
  uint32_T enginetorque_maxIndex[2];/* Computed Parameter: enginetorque_maxIndex
                                     * Referenced by: '<S5>/engine torque'
                                     */
};

/* Real-time Model Data Structure */
struct tag_RTM_TransmissionDownshiftTe {
  const char_T *errorStatus;
  RTWSolverInfo solverInfo;
  ContinuousStates_TransmissionDo *contStates;
  int_T *periodicContStateIndices;
  real_T *periodicContStateRanges;
  real_T *derivs;
  boolean_T *contStateDisabled;
  boolean_T zCCacheNeedsReset;
  boolean_T derivCacheNeedsReset;
  boolean_T CTOutputIncnstWithState;
  real_T odeF[1][2];
  ODE1_IntgData intgData;

  /*
   * Sizes:
   * The following substructure contains sizes information
   * for many of the model attributes such as inputs, outputs,
   * dwork, sample times, etc.
   */
  struct {
    int_T numContStates;
    int_T numPeriodicContStates;
    int_T numSampTimes;
  } Sizes;

  /*
   * Timing:
   * The following substructure contains information regarding
   * the timing information for the model.
   */
  struct {
    uint32_T clockTick0;
    uint32_T clockTickH0;
    time_T stepSize0;
    uint32_T clockTick1;
    uint32_T clockTickH1;
    struct {
      uint8_T TID[3];
    } TaskCounters;

    SimTimeStep simTimeStep;
    boolean_T stopRequestedFlag;
    time_T *t;
    time_T tArray[3];
  } Timing;
};

/* Block parameters (default storage) */
extern Parameters_TransmissionDownshif TransmissionDownshiftTestSequ_P;

/* Block signals (default storage) */
extern BlockIO_TransmissionDownshiftTe TransmissionDownshiftTestSequ_B;

/* Continuous states (default storage) */
extern ContinuousStates_TransmissionDo TransmissionDownshiftTestSequ_X;

/* Block states (default storage) */
extern D_Work_TransmissionDownshiftTes TransmissionDownshiftTest_DWork;

/* External inputs (root inport signals with default storage) */
extern ExternalInputs_TransmissionDown TransmissionDownshiftTestSequ_U;

/* External outputs (root outports fed by signals with default storage) */
extern ExternalOutputs_TransmissionDow TransmissionDownshiftTestSequ_Y;

/* Model entry point functions */
extern void TransmissionDownshiftTestSequence_initialize(void);
extern void TransmissionDownshiftTestSequence_output(void);
extern void TransmissionDownshiftTestSequence_update(void);
extern void TransmissionDownshiftTestSequence_terminate(void);

/* Real-time Model object */
extern RT_MODEL_TransmissionDownshiftT *const TransmissionDownshiftTestSeq_M;

/*-
 * The generated code includes comments that allow you to trace directly
 * back to the appropriate location in the model.  The basic format
 * is <system>/block_name, where system is the system number (uniquely
 * assigned by Simulink) and block_name is the name of the block.
 *
 * Use the MATLAB hilite_system command to trace the generated code back
 * to the model.  For example,
 *
 * hilite_system('<S3>')    - opens system 3
 * hilite_system('<S3>/Kp') - opens and selects block Kp which resides in S3
 *
 * Here is the system hierarchy for this model
 *
 * '<Root>' : 'TransmissionDownshiftTestSequence'
 * '<S1>'   : 'TransmissionDownshiftTestSequence/shift_controller'
 * '<S2>'   : 'TransmissionDownshiftTestSequence/vehicle'
 * '<S3>'   : 'TransmissionDownshiftTestSequence/shift_controller/selection_state.calc_th'
 * '<S4>'   : 'TransmissionDownshiftTestSequence/shift_controller/selection_state.calc_th/Look-Up'
 * '<S5>'   : 'TransmissionDownshiftTestSequence/vehicle/Engine'
 * '<S6>'   : 'TransmissionDownshiftTestSequence/vehicle/Vehicle'
 * '<S7>'   : 'TransmissionDownshiftTestSequence/vehicle/transmission'
 * '<S8>'   : 'TransmissionDownshiftTestSequence/vehicle/transmission/Torque Converter'
 * '<S9>'   : 'TransmissionDownshiftTestSequence/vehicle/transmission/transmission ratio'
 * '<S10>'  : 'TransmissionDownshiftTestSequence/vehicle/transmission/transmission ratio/Look-Up Table'
 */
#endif                     /* RTW_HEADER_TransmissionDownshiftTestSequence_h_ */
```

#### TransmissionDownshiftTestSequence_data.c
```c
/********************************************************************
 * COPYRIGHT -- Bernecker + Rainer Industrie-Elektronik Ges.m.b.H.
 ********************************************************************
 * Program: TransmissionDownshiftTestSequence
 * File: TransmissionDownshiftTestSequence_data.c
 * Author: The MathWorks, Inc.
 * Created: Wed Jun 03 01:12:01 1998
 ********************************************************************
 * Data for program TransmissionDownshiftTestSequence
 ********************************************************************
 * Generated with B&R Automation Studio Target for Simulink  V6.1.0
 * (ERT based)
 ********************************************************************/

#include "TransmissionDownshiftTestSequence.h"
#include "TransmissionDownshiftTestSequence_private.h"

/*  GLOBAL DATA DEFINITIONS */

/* Block parameters (default storage) */
Parameters_TransmissionDownshif TransmissionDownshiftTestSequ_P = {
  /* Variable: Iei
   * Referenced by: '<S5>/engine + impeller inertia'
   */
  0.021991488283555904,

  /* Variable: downtab
   * Referenced by: '<S3>/interp_down'
   */
  { 0.0, 0.0, 0.0, 0.0, 0.0, 0.0, 5.0, 5.0, 5.0, 5.0, 30.0, 30.0, 20.0, 20.0,
    25.0, 30.0, 50.0, 50.0, 35.0, 35.0, 40.0, 50.0, 80.0, 80.0 },

  /* Variable: downth
   * Referenced by: '<S3>/interp_down'
   */
  { 0.0, 5.0, 40.0, 50.0, 90.0, 100.0 },

  /* Variable: emap
   * Referenced by: '<S5>/engine torque'
   */
  { -40.0, 215.0, 245.0, 264.0, 264.0, 267.0, 267.0, 267.0, 267.0, 267.0, -44.0,
    117.0, 208.0, 260.0, 279.0, 290.0, 297.0, 301.0, 301.0, 301.0, -49.0, 85.0,
    178.0, 241.0, 282.0, 293.0, 305.0, 308.0, 312.0, 312.0, -53.0, 66.0, 148.0,
    219.0, 275.0, 297.0, 305.0, 312.0, 319.0, 319.0, -57.0, 44.0, 122.0, 193.0,
    260.0, 290.0, 305.0, 319.0, 327.0, 327.0, -61.0, 29.0, 104.0, 167.0, 238.0,
    275.0, 301.0, 323.0, 327.0, 334.0, -65.0, 10.0, 85.0, 152.0, 223.0, 260.0,
    293.0, 319.0, 327.0, 334.0, -70.0, -2.0, 66.0, 133.0, 208.0, 256.0, 282.0,
    316.0, 327.0, 334.0, -74.0, -13.0, 48.0, 119.0, 189.0, 234.0, 267.0, 297.0,
    312.0, 319.0, -78.0, -22.0, 33.0, 96.0, 171.0, 212.0, 249.0, 279.0, 293.0,
    305.0, -82.0, -32.0, 18.0, 85.0, 152.0, 193.0, 226.0, 253.0, 267.0, 275.0 },

  /* Variable: nevec
   * Referenced by: '<S5>/engine torque'
   */
  { 799.99999999999989, 1200.0, 1599.9999999999998, 1999.9999999999998, 2400.0,
    2800.0000000000005, 3199.9999999999995, 3599.9999999999995,
    3999.9999999999995, 4400.0, 4800.0 },

  /* Variable: thvec
   * Referenced by: '<S5>/engine torque'
   */
  { 0.0, 20.0, 30.0, 40.0, 50.0, 60.0, 70.0, 80.0, 90.0, 100.0 },

  /* Variable: uptab
   * Referenced by: '<S3>/interp_up'
   */
  { 10.0, 10.0, 15.0, 23.0, 40.0, 40.0, 30.0, 30.0, 30.0, 41.0, 70.0, 70.0, 50.0,
    50.0, 50.0, 60.0, 100.0, 100.0, 1.0E+6, 1.0E+6, 1.0E+6, 1.0E+6, 1.0E+6,
    1.0E+6 },

  /* Variable: upth
   * Referenced by: '<S3>/interp_up'
   */
  { 0.0, 25.0, 35.0, 50.0, 90.0, 100.0 },

  /* Variable: vehicledata
   * Referenced by:
   *   '<S6>/final drive ratio1'
   *   '<S6>/final drive ratio2'
   *   '<S6>/linear speed'
   *   '<S6>/vehicle inertia'
   *   '<S6>/wheel speed'
   */
  { 3.23, 40.0, 0.3, 1.0, 50.0, 0.0 },

  /* Mask Parameter: TorqueConverter_Kfactor
   * Referenced by: '<S8>/K factor'
   */
  { 137.4652089938063, 137.06501915685197, 135.86444964598905,
    135.66435472751189, 137.56525645304487, 140.36658531172509,
    145.26891081441539, 152.87251771654735, 162.97731109964374,
    164.2779280697452, 166.17882979527823, 167.97968406157264,
    170.08068070558275, 172.78196210502438, 175.38319604522741,
    179.58518933324765, 183.58708770279083, 189.89007763482121,
    197.69377945543027, 215.90241703685155, 244.51599037908485 },

  /* Mask Parameter: TorqueConverter_Torkratio
   * Referenced by: '<S8>/Torque ratio'
   */
  { 2.2319999999999998, 2.075, 1.975, 1.8459999999999999, 1.72, 1.564, 1.409,
    1.254, 1.0959999999999999, 1.08, 1.061, 1.043, 1.028, 1.012, 1.002, 1.002,
    1.001, 0.998, 0.99900000000000011, 1.001, 1.002 },

  /* Mask Parameter: TorqueConverter_speedratio
   * Referenced by:
   *   '<S8>/K factor'
   *   '<S8>/Torque ratio'
   */
  { 0.0, 0.1, 0.2, 0.30000000000000004, 0.4, 0.5, 0.60000000000000009,
    0.70000000000000007, 0.8, 0.81, 0.82000000000000006, 0.83000000000000007,
    0.84, 0.85, 0.86, 0.87, 0.88, 0.89, 0.9, 0.92, 0.94 },

  /* Mask Parameter: shift_controller_TWAIT
   * Referenced by: '<Root>/shift_controller'
   */
  2U,

  /* Expression: [1:4]
   * Referenced by: '<S3>/interp_down'
   */
  { 1.0, 2.0, 3.0, 4.0 },

  /* Expression: [1:4]
   * Referenced by: '<S3>/interp_up'
   */
  { 1.0, 2.0, 3.0, 4.0 },

  /* Expression: 60/5280
   * Referenced by: '<S6>/mph'
   */
  0.011363636363636364,

  /* Expression: 1000
   * Referenced by: '<S5>/Integrator'
   */
  1000.0,

  /* Expression: 6000
   * Referenced by: '<S5>/Integrator'
   */
  6000.0,

  /* Expression: 600
   * Referenced by: '<S5>/Integrator'
   */
  600.0,

  /* Computed Parameter: interp_down_maxIndex
   * Referenced by: '<S3>/interp_down'
   */
  { 5U, 3U },

  /* Computed Parameter: interp_up_maxIndex
   * Referenced by: '<S3>/interp_up'
   */
  { 5U, 3U },

  /* Computed Parameter: enginetorque_maxIndex
   * Referenced by: '<S5>/engine torque'
   */
  { 9U, 10U }
};
```

#### TransmissionDownshiftTestSequence_private.h
```c
/********************************************************************
 * COPYRIGHT -- Bernecker + Rainer Industrie-Elektronik Ges.m.b.H.
 ********************************************************************
 * Program: TransmissionDownshiftTestSequence
 * File: TransmissionDownshiftTestSequence_private.h
 * Author: The MathWorks, Inc.
 * Created: Wed Jun 03 01:12:01 1998
 ********************************************************************
 * Header for program TransmissionDownshiftTestSequence
 ********************************************************************
 * Generated with B&R Automation Studio Target for Simulink  V6.1.0
 * (ERT based)
 ********************************************************************/

#ifndef RTW_HEADER_TransmissionDownshiftTestSequence_private_h_
#define RTW_HEADER_TransmissionDownshiftTestSequence_private_h_
#include "rtwtypes.h"
#define _ASMATH_
#define ASMATH_
#define _ASMATH_H
#define ASMATH_H
#define _ASMATH_H_
#define ASMATH_H_
#define _ASSTRING_
#define ASSTRING_
#define _ASSTRING_H
#define ASSTRING_H
#define _ASSTRING_H_
#define ASSTRING_H_
#include <bur/plctypes.h>
#ifdef _DEFAULT_INCLUDES
#include <AsDefault.h>
#endif

/* Private macros used by the generated code to access rtModel */
#ifndef rtmIsMajorTimeStep
# define rtmIsMajorTimeStep(rtm)       (((rtm)->Timing.simTimeStep) == MAJOR_TIME_STEP)
#endif

#ifndef rtmIsMinorTimeStep
# define rtmIsMinorTimeStep(rtm)       (((rtm)->Timing.simTimeStep) == MINOR_TIME_STEP)
#endif

#ifndef rtmSetTPtr
# define rtmSetTPtr(rtm, val)          ((rtm)->Timing.t = (val))
#endif

#ifndef MIN
#define MIN(a,b)                       ((a) < (b) ? (a) : (b))
#endif

#ifndef MAX
#define MAX(a,b)                       ((a) > (b) ? (a) : (b))
#endif

extern real_T look1_binlxpw(real_T u0, const real_T bp0[], const real_T table[],
  uint32_T maxIndex);
extern real_T look2_binlxpw(real_T u0, real_T u1, const real_T bp0[], const
  real_T bp1[], const real_T table[], const uint32_T maxIndex[], uint32_T stride);

/* private model entry point functions */
extern void TransmissionDownshiftTestSequence_derivatives(void);

#endif             /* RTW_HEADER_TransmissionDownshiftTestSequence_private_h_ */
```

#### TransmissionDownshiftTestSequence_types.h
```c
/********************************************************************
 * COPYRIGHT -- Bernecker + Rainer Industrie-Elektronik Ges.m.b.H.
 ********************************************************************
 * Program: TransmissionDownshiftTestSequence
 * File: TransmissionDownshiftTestSequence_types.h
 * Author: The MathWorks, Inc.
 * Created: Wed Jun 03 01:12:01 1998
 ********************************************************************
 * Header for program TransmissionDownshiftTestSequence
 ********************************************************************
 * Generated with B&R Automation Studio Target for Simulink  V6.1.0
 * (ERT based)
 ********************************************************************/

#ifndef RTW_HEADER_TransmissionDownshiftTestSequence_types_h_
#define RTW_HEADER_TransmissionDownshiftTestSequence_types_h_
#include "rtwtypes.h"
#ifndef MIN
#define MIN(a,b)                       ((a) < (b) ? (a) : (b))
#endif

#ifndef MAX
#define MAX(a,b)                       ((a) > (b) ? (a) : (b))
#endif

#ifndef DEFINED_TYPEDEF_FOR_gearType_
#define DEFINED_TYPEDEF_FOR_gearType_

typedef enum {
  gearType_None = 0,                   /* Default value */
  gearType_first,
  gearType_second,
  gearType_third,
  gearType_fourth
} gearType;

#endif

/* Parameters (default storage) */
typedef struct Parameters_TransmissionDownshif_ Parameters_TransmissionDownshif;

/* Forward declaration for rtModel */
typedef struct tag_RTM_TransmissionDownshiftTe RT_MODEL_TransmissionDownshiftT;

#endif               /* RTW_HEADER_TransmissionDownshiftTestSequence_types_h_ */
```

#### rtwtypes.h
```c
/********************************************************************
 * COPYRIGHT -- Bernecker + Rainer Industrie-Elektronik Ges.m.b.H.
 ********************************************************************
 * Program: TransmissionDownshiftTestSequence
 * File: rtwtypes.h
 * Author: The MathWorks, Inc.
 * Created: Wed Jun 03 01:12:01 1998
 ********************************************************************
 * Header for program TransmissionDownshiftTestSequence
 ********************************************************************
 * Generated with B&R Automation Studio Target for Simulink  V6.1.0
 * (ERT based)
 ********************************************************************/

#ifndef RTWTYPES_H
#define RTWTYPES_H

/* Logical type definitions */
#if (!defined(__cplusplus))
#  ifndef false
#   define false                       (0U)
#  endif

#  ifndef true
#   define true                        (1U)
#  endif
#endif

/*=======================================================================*
 * Target hardware information
 *   Device type: Intel->x86/Pentium
 *   Number of bits:     char:   8    short:   16    long:  32
 *                       long:  32
 *                       native word size:  32
 *   Byte ordering: LittleEndian
 *   Signed integer division rounds to: Zero
 *   Shift right on a signed integer as arithmetic shift: on
 *=======================================================================*/

/*=======================================================================*
 * Fixed width word size data types:                                     *
 *   int8_T, int16_T, int32_T     - signed 8, 16, or 32 bit integers     *
 *   uint8_T, uint16_T, uint32_T  - unsigned 8, 16, or 32 bit integers   *
 *   real32_T, real64_T           - 32 and 64 bit floating point numbers *
 *=======================================================================*/
typedef signed char int8_T;
typedef unsigned char uint8_T;
typedef short int16_T;
typedef unsigned short uint16_T;
typedef long int32_T;
typedef unsigned long uint32_T;
typedef float real32_T;
typedef double real64_T;

/*===========================================================================*
 * Generic type definitions: boolean_T, char_T, byte_T, int_T, uint_T,       *
 *                           real_T, time_T, ulong_T.                        *
 *===========================================================================*/
typedef double real_T;
typedef double time_T;
typedef unsigned char boolean_T;
typedef long int_T;
typedef unsigned long uint_T;
typedef unsigned long ulong_T;
typedef char char_T;
typedef unsigned char uchar_T;
typedef char_T byte_T;

/*===========================================================================*
 * Complex number type definitions                                           *
 *===========================================================================*/
#define CREAL_T

typedef struct {
  real32_T re;
  real32_T im;
} creal32_T;

typedef struct {
  real64_T re;
  real64_T im;
} creal64_T;

typedef struct {
  real_T re;
  real_T im;
} creal_T;

#define CINT8_T

typedef struct {
  int8_T re;
  int8_T im;
} cint8_T;

#define CUINT8_T

typedef struct {
  uint8_T re;
  uint8_T im;
} cuint8_T;

#define CINT16_T

typedef struct {
  int16_T re;
  int16_T im;
} cint16_T;

#define CUINT16_T

typedef struct {
  uint16_T re;
  uint16_T im;
} cuint16_T;

#define CINT32_T

typedef struct {
  int32_T re;
  int32_T im;
} cint32_T;

#define CUINT32_T

typedef struct {
  uint32_T re;
  uint32_T im;
} cuint32_T;

/*=======================================================================*
 * Min and Max:                                                          *
 *   int8_T, int16_T, int32_T     - signed 8, 16, or 32 bit integers     *
 *   uint8_T, uint16_T, uint32_T  - unsigned 8, 16, or 32 bit integers   *
 *=======================================================================*/
#define MAX_int8_T                     ((int8_T)(127))
#define MIN_int8_T                     ((int8_T)(-128))
#define MAX_uint8_T                    ((uint8_T)(255U))
#define MAX_int16_T                    ((int16_T)(32767))
#define MIN_int16_T                    ((int16_T)(-32768))
#define MAX_uint16_T                   ((uint16_T)(65535U))
#define MAX_int32_T                    ((int32_T)(2147483647))
#define MIN_int32_T                    ((int32_T)(-2147483647-1))
#define MAX_uint32_T                   ((uint32_T)(0xFFFFFFFFU))

/* Block D-Work pointer type */
typedef void * pointer_T;

#endif                                 /* RTWTYPES_H */

#ifndef MIN
#define MIN(a,b)                       ((a) < (b) ? (a) : (b))
#endif

#ifndef MAX
#define MAX(a,b)                       ((a) > (b) ? (a) : (b))
#endif
```

#### task_properties.txt
```
For manual assignment to hardware configuration please
add the following additional include directories:

\Logical\MATLAB_includes\R2019b\

And the following additional build options:

-lm -D MODEL=TransmissionDownshiftTestSequence -D NUMST=3 -D NCSTATES=2 -D HAVESTDIO -D MODEL_HAS_DYNAMICALLY_LOADED_SFCNS=0 -D CLASSIC_INTERFACE=0 -D ALLOCATIONFCN=0 -D TID01EQ=1 -D TERMFCN=1 -D ONESTEPFCN=0 -D MAT_FILE=0 -D MULTI_INSTANCE_CODE=0 -D INTEGER_CODE=0 -D MT=0
```

### Program Logical/sltest (ANSIC, version 1.00.0)

#### sltest.var
```iecst
VAR
	    Active_Control : BOOL := 0; (**)
END_VAR
```

#### rtwtypes.h
```c
/********************************************************************
 * COPYRIGHT -- Bernecker + Rainer Industrie-Elektronik Ges.m.b.H.
 ********************************************************************
 * Program: sltestCruiseControlDefective
 * File: rtwtypes.h
 * Author: The MathWorks, Inc.
 * Created: Wed Aug 30 21:41:02 2006
 ********************************************************************
 * Header for program sltestCruiseControlDefective
 ********************************************************************
 * Generated with B&R Automation Studio Target for Simulink  V6.1.0
 * (ERT based)
 ********************************************************************/

#ifndef RTWTYPES_H
#define RTWTYPES_H

/* Logical type definitions */
#if (!defined(__cplusplus))
#  ifndef false
#   define false                       (0U)
#  endif

#  ifndef true
#   define true                        (1U)
#  endif
#endif

/*=======================================================================*
 * Target hardware information
 *   Device type: Intel->x86/Pentium
 *   Number of bits:     char:   8    short:   16    long:  32
 *                       long:  32
 *                       native word size:  32
 *   Byte ordering: LittleEndian
 *   Signed integer division rounds to: Zero
 *   Shift right on a signed integer as arithmetic shift: on
 *=======================================================================*/

/*=======================================================================*
 * Fixed width word size data types:                                     *
 *   int8_T, int16_T, int32_T     - signed 8, 16, or 32 bit integers     *
 *   uint8_T, uint16_T, uint32_T  - unsigned 8, 16, or 32 bit integers   *
 *   real32_T, real64_T           - 32 and 64 bit floating point numbers *
 *=======================================================================*/
typedef signed char int8_T;
typedef unsigned char uint8_T;
typedef short int16_T;
typedef unsigned short uint16_T;
typedef long int32_T;
typedef unsigned long uint32_T;
typedef float real32_T;
typedef double real64_T;

/*===========================================================================*
 * Generic type definitions: boolean_T, char_T, byte_T, int_T, uint_T,       *
 *                           real_T, time_T, ulong_T.                        *
 *===========================================================================*/
typedef double real_T;
typedef double time_T;
typedef unsigned char boolean_T;
typedef long int_T;
typedef unsigned long uint_T;
typedef unsigned long ulong_T;
typedef char char_T;
typedef unsigned char uchar_T;
typedef char_T byte_T;

/*===========================================================================*
 * Complex number type definitions                                           *
 *===========================================================================*/
#define CREAL_T

typedef struct {
  real32_T re;
  real32_T im;
} creal32_T;

typedef struct {
  real64_T re;
  real64_T im;
} creal64_T;

typedef struct {
  real_T re;
  real_T im;
} creal_T;

#define CINT8_T

typedef struct {
  int8_T re;
  int8_T im;
} cint8_T;

#define CUINT8_T

typedef struct {
  uint8_T re;
  uint8_T im;
} cuint8_T;

#define CINT16_T

typedef struct {
  int16_T re;
  int16_T im;
} cint16_T;

#define CUINT16_T

typedef struct {
  uint16_T re;
  uint16_T im;
} cuint16_T;

#define CINT32_T

typedef struct {
  int32_T re;
  int32_T im;
} cint32_T;

#define CUINT32_T

typedef struct {
  uint32_T re;
  uint32_T im;
} cuint32_T;

/*=======================================================================*
 * Min and Max:                                                          *
 *   int8_T, int16_T, int32_T     - signed 8, 16, or 32 bit integers     *
 *   uint8_T, uint16_T, uint32_T  - unsigned 8, 16, or 32 bit integers   *
 *=======================================================================*/
#define MAX_int8_T                     ((int8_T)(127))
#define MIN_int8_T                     ((int8_T)(-128))
#define MAX_uint8_T                    ((uint8_T)(255U))
#define MAX_int16_T                    ((int16_T)(32767))
#define MIN_int16_T                    ((int16_T)(-32768))
#define MAX_uint16_T                   ((uint16_T)(65535U))
#define MAX_int32_T                    ((int32_T)(2147483647))
#define MIN_int32_T                    ((int32_T)(-2147483647-1))
#define MAX_uint32_T                   ((uint32_T)(0xFFFFFFFFU))

/* Block D-Work pointer type */
typedef void * pointer_T;

#endif                                 /* RTWTYPES_H */

#ifndef MIN
#define MIN(a,b)                       ((a) < (b) ? (a) : (b))
#endif

#ifndef MAX
#define MAX(a,b)                       ((a) > (b) ? (a) : (b))
#endif
```

#### sltest.c
```c
/********************************************************************
 * COPYRIGHT -- Bernecker + Rainer Industrie-Elektronik Ges.m.b.H.
 ********************************************************************
 * Program: sltestCruiseControlDefective
 * File: sltest.c
 * Author: The MathWorks, Inc.
 * Created: Wed Aug 30 21:41:02 2006
 ********************************************************************
 * Implementation of program sltestCruiseControlDefective
 ********************************************************************
 * Generated with B&R Automation Studio Target for Simulink  V6.1.0
 * (ERT based)
 ********************************************************************/

#define _ASMATH_
#define ASMATH_
#define _ASMATH_H
#define ASMATH_H
#define _ASMATH_H_
#define ASMATH_H_
#define _ASSTRING_
#define ASSTRING_
#define _ASSTRING_H
#define ASSTRING_H
#define _ASSTRING_H_
#define ASSTRING_H_
#include <bur/plctypes.h>
#ifdef _DEFAULT_INCLUDES
#include <AsDefault.h>
#endif

#include "sltestCruiseControlDefective.h"
#include "rtwtypes.h"

/*  Defines */

/*  Data Types */

/**************************** GLOBAL DATA *************************************/
/*  Definitions */

/*  Declarations  */

/***************************** FILE SCOPE DATA ********************************/

/*************************** FUNCTIONS ****************************************/
#ifdef __cplusplus

unsigned long bur_heap_size = 6553500;

#endif

  void _INIT mainINIT(void)
{

    UDINT st_ident;
  RTInfo_typ rt_info;
  rt_info.enable = 1;
  RTInfo(&rt_info);
  if (rt_info.cycle_time != 10000) {
    /* cycle time does not match Simulink fixed-step size */
    ST_ident("sltest", 0, &st_ident);
    ST_tmp_suspend(st_ident);
    ERR_warning(33310, 0);
  }

  /* initialize model */
  sltestCruiseControlDefective_initialize();

} void _CYCLIC mainCYCLIC(void)
{
  /* call model step function */
  sltestCruiseControlDefective_output();

  sltestCruiseControlDefective_update();

} void _EXIT mainEXIT(void)
{
  /* terminate model */
  sltestCruiseControlDefective_terminate();

} /*****************************************************************************
     Task sample time: 0.01s
   *****************************************************************************/
/*****************************************************************************
   B&R Automation Studio Target for Simulink Version: V6.1.0 (06-Nov-2019)
 *****************************************************************************/

/*======================== TOOL VERSION INFORMATION ==========================*
 * MATLAB 9.7 (R2019b)18-Jul-2019                                             *
 * Simulink 10.0 (R2019b)18-Jul-2019                                          *
 * Simulink Coder 9.2 (R2019b)18-Jul-2019                                     *
 * Embedded Coder 7.3 (R2019b)18-Jul-2019                                     *
 * Stateflow 10.1 (R2019b)18-Jul-2019                                         *
 * Fixed-Point Designer 6.4 (R2019b)18-Jul-2019                               *
 *============================================================================*/

/*======================= LICENSE IN USE INFORMATION =========================*
 * matlab                                                                     *
 * matlab_coder                                                               *
 * real-time_workshop                                                         *
 * rtw_embedded_coder                                                         *
 * simulink                                                                   *
 * simulink_test                                                              *
 * stateflow                                                                  *
 *============================================================================*/
```

#### sltestCruiseControlDefective.c
```c
/********************************************************************
 * COPYRIGHT -- Bernecker + Rainer Industrie-Elektronik Ges.m.b.H.
 ********************************************************************
 * Program: sltestCruiseControlDefective
 * File: sltestCruiseControlDefective.c
 * Author: The MathWorks, Inc.
 * Created: Wed Aug 30 21:41:02 2006
 ********************************************************************
 * Implementation of program sltestCruiseControlDefective
 ********************************************************************
 * Generated with B&R Automation Studio Target for Simulink  V6.1.0
 * (ERT based)
 ********************************************************************/

#include "sltestCruiseControlDefective.h"
#include "sltestCruiseControlDefective_private.h"

/*  Defines */

/*  Data Types */

/**************************** GLOBAL DATA *************************************/
/*  Definitions */

/* Block signals (default storage) */
BlockIO_sltestCruiseControlDefe sltestCruiseControlDefective_B;

/* Block states (default storage) */
D_Work_sltestCruiseControlDefec sltestCruiseControlDefect_DWork;

/* External outputs (root outports fed by signals with default storage) */
ExternalOutputs_sltestCruiseCon sltestCruiseControlDefective_Y;

/* Real-time model */
RT_MODEL_sltestCruiseControlDef sltestCruiseControlDefective_M_;
RT_MODEL_sltestCruiseControlDef *const sltestCruiseControlDefective_M =
  &sltestCruiseControlDefective_M_;

/*  Declarations  */

/***************************** FILE SCOPE DATA ********************************/

/*************************** FUNCTIONS ****************************************/

/* Model output function */
void sltestCruiseControlDefective_output(void)
{
  /* local block i/o variables */
  real_T rtb_FromWs[6];

  /* FromWorkspace: '<S2>/FromWs' */
  {
    real_T *pDataValues = (real_T *)
      sltestCruiseControlDefect_DWork.FromWs_PWORK.DataPtr;
    real_T *pTimeValues = (real_T *)
      sltestCruiseControlDefect_DWork.FromWs_PWORK.TimePtr;
    int_T currTimeIndex = sltestCruiseControlDefect_DWork.FromWs_IWORK.PrevIndex;
    real_T t = sltestCruiseControlDefective_M->Timing.t[0];

    /* Get index */
    if (t <= pTimeValues[0]) {
      currTimeIndex = 0;
    } else if (t >= pTimeValues[105]) {
      currTimeIndex = 104;
    } else {
      if (t < pTimeValues[currTimeIndex]) {
        while (t < pTimeValues[currTimeIndex]) {
          currTimeIndex--;
        }
      } else {
        while (t >= pTimeValues[currTimeIndex + 1]) {
          currTimeIndex++;
        }
      }
    }

    sltestCruiseControlDefect_DWork.FromWs_IWORK.PrevIndex = currTimeIndex;

    /* Post output */
    {
      real_T t1 = pTimeValues[currTimeIndex];
      real_T t2 = pTimeValues[currTimeIndex + 1];
      if (t1 == t2) {
        if (t < t1) {
          {
            int_T elIdx;
            for (elIdx = 0; elIdx < 6; ++elIdx) {
              (&rtb_FromWs[0])[elIdx] = pDataValues[currTimeIndex];
              pDataValues += 106;
            }
          }
        } else {
          {
            int_T elIdx;
            for (elIdx = 0; elIdx < 6; ++elIdx) {
              (&rtb_FromWs[0])[elIdx] = pDataValues[currTimeIndex + 1];
              pDataValues += 106;
            }
          }
        }
      } else {
        real_T f1 = (t2 - t) / (t2 - t1);
        real_T f2 = 1.0 - f1;
        real_T d1;
        real_T d2;
        int_T TimeIndex= currTimeIndex;

        {
          int_T elIdx;
          for (elIdx = 0; elIdx < 6; ++elIdx) {
            d1 = pDataValues[TimeIndex];
            d2 = pDataValues[TimeIndex + 1];
            (&rtb_FromWs[0])[elIdx] = (real_T) rtInterpolate(d1, d2, f1, f2);
            pDataValues += 106;
          }
        }
      }
    }
  }

  /* Switch: '<S1>/Switch1' incorporates:
   *  DataTypeConversion: '<S4>/Cast4'
   *  DataTypeConversion: '<S4>/Cast5'
   *  DataTypeConversion: '<S4>/Cast6'
   *  Switch: '<S1>/Switch2'
   *  Switch: '<S1>/Switch3'
   */
  if (rtb_FromWs[3] != 0.0) {
    /* Outport: '<Root>/target' incorporates:
     *  DataTypeConversion: '<S4>/Cast1'
     */
    sltestCruiseControlDefective_Y.target = rtb_FromWs[0];
  } else if (rtb_FromWs[4] != 0.0) {
    /* Switch: '<S1>/Switch2' incorporates:
     *  Constant: '<S1>/Constant1'
     *  Outport: '<Root>/target'
     *  Sum: '<S1>/Sum'
     *  UnitDelay: '<S1>/Unit Delay'
     */
    sltestCruiseControlDefective_Y.target =
      sltestCruiseControlDefective_P.Constant1_Value +
      sltestCruiseControlDefect_DWork.UnitDelay_DSTATE;
  } else if (rtb_FromWs[5] != 0.0) {
    /* Switch: '<S1>/Switch3' incorporates:
     *  Constant: '<S1>/Constant3'
     *  Outport: '<Root>/target'
     *  Sum: '<S1>/Sum2'
     *  Switch: '<S1>/Switch2'
     *  UnitDelay: '<S1>/Unit Delay'
     */
    sltestCruiseControlDefective_Y.target =
      sltestCruiseControlDefect_DWork.UnitDelay_DSTATE -
      sltestCruiseControlDefective_P.Constant3_Value;
  } else {
    /* Outport: '<Root>/target' incorporates:
     *  Switch: '<S1>/Switch2'
     *  Switch: '<S1>/Switch3'
     *  UnitDelay: '<S1>/Unit Delay'
     */
    sltestCruiseControlDefective_Y.target =
      sltestCruiseControlDefect_DWork.UnitDelay_DSTATE;
  }

  /* End of Switch: '<S1>/Switch1' */

  /* Sum: '<S1>/Sum1' incorporates:
   *  DataTypeConversion: '<S4>/Cast1'
   *  Outport: '<Root>/target'
   */
  sltestCruiseControlDefective_B.Sum1 = sltestCruiseControlDefective_Y.target -
    rtb_FromWs[0];

  /* Logic: '<S1>/Logical Operator' incorporates:
   *  DataTypeConversion: '<S4>/Cast2'
   *  DataTypeConversion: '<S4>/Cast3'
   *  DataTypeConversion: '<S4>/Cast4'
   *  Logic: '<S1>/Logical Operator1'
   *  Logic: '<S1>/Logical Operator2'
   *  UnitDelay: '<S1>/Unit Delay1'
   */
  sltestCruiseControlDefective_B.ActiveControl = ((rtb_FromWs[1] != 0.0) &&
    (rtb_FromWs[2] == 0.0) && ((rtb_FromWs[3] != 0.0) ||
    sltestCruiseControlDefect_DWork.UnitDelay1_DSTATE));

  /* Outputs for Enabled SubSystem: '<S1>/PI Controller' incorporates:
   *  EnablePort: '<S5>/Enable'
   */
  if (sltestCruiseControlDefective_B.ActiveControl) {
    /* Outport: '<Root>/throt' incorporates:
     *  DiscreteIntegrator: '<S5>/Discrete-Time Integrator'
     *  Gain: '<S5>/Kp'
     *  Gain: '<S5>/Kp1'
     *  Sum: '<S5>/Sum'
     */
    sltestCruiseControlDefective_Y.throt =
      sltestCruiseControlDefective_P.Kp_Gain *
      sltestCruiseControlDefective_B.Sum1 +
      sltestCruiseControlDefective_P.Kp1_Gain *
      sltestCruiseControlDefect_DWork.DiscreteTimeIntegrator_DSTATE;
  }

  /* End of Outputs for SubSystem: '<S1>/PI Controller' */

  /* S-Function (bur_out): '<S1>/Output' */
  Active_Control = sltestCruiseControlDefective_B.ActiveControl;
}

/* Model update function */
void sltestCruiseControlDefective_update(void)
{
  /* Update for UnitDelay: '<S1>/Unit Delay' incorporates:
   *  Outport: '<Root>/target'
   */
  sltestCruiseControlDefect_DWork.UnitDelay_DSTATE =
    sltestCruiseControlDefective_Y.target;

  /* Update for UnitDelay: '<S1>/Unit Delay1' */
  sltestCruiseControlDefect_DWork.UnitDelay1_DSTATE =
    sltestCruiseControlDefective_B.ActiveControl;

  /* Update for Enabled SubSystem: '<S1>/PI Controller' incorporates:
   *  EnablePort: '<S5>/Enable'
   */
  if (sltestCruiseControlDefective_B.ActiveControl) {
    /* Update for DiscreteIntegrator: '<S5>/Discrete-Time Integrator' */
    sltestCruiseControlDefect_DWork.DiscreteTimeIntegrator_DSTATE +=
      sltestCruiseControlDefective_P.DiscreteTimeIntegrator_gainval *
      sltestCruiseControlDefective_B.Sum1;
    if (sltestCruiseControlDefect_DWork.DiscreteTimeIntegrator_DSTATE >=
        sltestCruiseControlDefective_P.DiscreteTimeIntegrator_UpperSat) {
      sltestCruiseControlDefect_DWork.DiscreteTimeIntegrator_DSTATE =
        sltestCruiseControlDefective_P.DiscreteTimeIntegrator_UpperSat;
    } else {
      if (sltestCruiseControlDefect_DWork.DiscreteTimeIntegrator_DSTATE <=
          sltestCruiseControlDefective_P.DiscreteTimeIntegrator_LowerSat) {
        sltestCruiseControlDefect_DWork.DiscreteTimeIntegrator_DSTATE =
          sltestCruiseControlDefective_P.DiscreteTimeIntegrator_LowerSat;
      }
    }

    /* End of Update for DiscreteIntegrator: '<S5>/Discrete-Time Integrator' */
  }

  /* End of Update for SubSystem: '<S1>/PI Controller' */

  /* Update absolute time for base rate */
  /* The "clockTick0" counts the number of times the code of this task has
   * been executed. The absolute time is the multiplication of "clockTick0"
   * and "Timing.stepSize0". Size of "clockTick0" ensures timer will not
   * overflow during the application lifespan selected.
   * Timer of this task consists of two 32 bit unsigned integers.
   * The two integers represent the low bits Timing.clockTick0 and the high bits
   * Timing.clockTickH0. When the low bit overflows to 0, the high bits increment.
   */
  if (!(++sltestCruiseControlDefective_M->Timing.clockTick0)) {
    ++sltestCruiseControlDefective_M->Timing.clockTickH0;
  }

  sltestCruiseControlDefective_M->Timing.t[0] =
    sltestCruiseControlDefective_M->Timing.clockTick0 *
    sltestCruiseControlDefective_M->Timing.stepSize0 +
    sltestCruiseControlDefective_M->Timing.clockTickH0 *
    sltestCruiseControlDefective_M->Timing.stepSize0 * 4294967296.0;

  {
    /* Update absolute timer for sample time: [0.01s, 0.0s] */
    /* The "clockTick1" counts the number of times the code of this task has
     * been executed. The resolution of this integer timer is 0.01, which is the step size
     * of the task. Size of "clockTick1" ensures timer will not overflow during the
     * application lifespan selected.
     * Timer of this task consists of two 32 bit unsigned integers.
     * The two integers represent the low bits Timing.clockTick1 and the high bits
     * Timing.clockTickH1. When the low bit overflows to 0, the high bits increment.
     */
    sltestCruiseControlDefective_M->Timing.clockTick1++;
    if (!sltestCruiseControlDefective_M->Timing.clockTick1) {
      sltestCruiseControlDefective_M->Timing.clockTickH1++;
    }
  }
}

/* Model initialize function */
void sltestCruiseControlDefective_initialize(void)
{
  /* Registration code */
  {
    /* Setup solver object */
    rtsiSetSimTimeStepPtr(&sltestCruiseControlDefective_M->solverInfo,
                          &sltestCruiseControlDefective_M->Timing.simTimeStep);
    rtsiSetTPtr(&sltestCruiseControlDefective_M->solverInfo, &rtmGetTPtr
                (sltestCruiseControlDefective_M));
    rtsiSetStepSizePtr(&sltestCruiseControlDefective_M->solverInfo,
                       &sltestCruiseControlDefective_M->Timing.stepSize0);
    rtsiSetErrorStatusPtr(&sltestCruiseControlDefective_M->solverInfo,
                          (&rtmGetErrorStatus(sltestCruiseControlDefective_M)));
    rtsiSetRTModelPtr(&sltestCruiseControlDefective_M->solverInfo,
                      sltestCruiseControlDefective_M);
  }

  rtsiSetSimTimeStep(&sltestCruiseControlDefective_M->solverInfo,
                     MAJOR_TIME_STEP);
  rtsiSetSolverName(&sltestCruiseControlDefective_M->solverInfo,
                    "FixedStepDiscrete");
  rtmSetTPtr(sltestCruiseControlDefective_M,
             &sltestCruiseControlDefective_M->Timing.tArray[0]);
  sltestCruiseControlDefective_M->Timing.stepSize0 = 0.01;

  /* Start for FromWorkspace: '<S2>/FromWs' */
  {
    static real_T pTimeValues0[] = { 0.0, 0.01, 0.01, 0.02, 0.02, 0.03, 0.03,
      0.04, 0.05, 0.06, 0.07, 0.08, 0.09, 0.1, 0.11, 0.12, 0.13, 0.14, 0.15,
      0.16, 0.17, 0.18, 0.19, 0.2, 0.2, 0.21, 0.21, 0.22, 0.23, 0.24, 0.25, 0.26,
      0.27, 0.28, 0.29, 0.3, 0.31, 0.32, 0.33, 0.34, 0.35, 0.36, 0.37, 0.38,
      0.39, 0.4, 0.41, 0.42, 0.43, 0.44, 0.45, 0.46, 0.47, 0.48, 0.49, 0.5, 0.51,
      0.52, 0.53, 0.54, 0.55, 0.56, 0.57, 0.58, 0.59, 0.6, 0.61, 0.62, 0.63,
      0.64, 0.65, 0.66, 0.67, 0.68, 0.69, 0.7, 0.71, 0.72, 0.73, 0.74, 0.75,
      0.76, 0.77, 0.78, 0.79, 0.8, 0.81, 0.82, 0.83, 0.84, 0.85, 0.86, 0.87,
      0.88, 0.89, 0.9, 0.91, 0.92, 0.93, 0.94, 0.95, 0.96, 0.97, 0.98, 0.99, 1.0
    } ;

    static real_T pDataValues0[] = { 40.0, 40.0, 40.0, 40.0, 40.0, 40.0, 40.0,
      40.0, 40.0, 40.0, 40.0, 40.0, 40.0, 40.0, 40.0, 40.0, 40.0, 40.0, 40.0,
      40.0, 40.0, 40.0, 40.0, 40.0, 40.0, 40.0, 40.0, 40.0, 40.0, 40.0, 40.0,
      40.0, 40.0, 40.0, 40.0, 40.0, 40.0, 40.0, 40.0, 40.0, 40.0, 40.0, 40.0,
      40.0, 40.0, 40.0, 40.0, 40.0, 40.0, 40.0, 40.0, 40.0, 40.0, 40.0, 40.0,
      40.0, 40.0, 40.0, 40.0, 40.0, 40.0, 40.0, 40.0, 40.0, 40.0, 40.0, 40.0,
      40.0, 40.0, 40.0, 40.0, 40.0, 40.0, 40.0, 40.0, 40.0, 40.0, 40.0, 40.0,
      40.0, 40.0, 40.0, 40.0, 40.0, 40.0, 40.0, 40.0, 40.0, 40.0, 40.0, 40.0,
      40.0, 40.0, 40.0, 40.0, 40.0, 40.0, 40.0, 40.0, 40.0, 40.0, 40.0, 40.0,
      40.0, 40.0, 40.0, 1.0, 1.0, 1.0, 1.0, 1.0, 1.0, 1.0, 1.0, 1.0, 1.0, 1.0,
      1.0, 1.0, 1.0, 1.0, 1.0, 1.0, 1.0, 1.0, 1.0, 1.0, 1.0, 1.0, 1.0, 1.0, 1.0,
      1.0, 1.0, 1.0, 1.0, 1.0, 1.0, 1.0, 1.0, 1.0, 1.0, 1.0, 1.0, 1.0, 1.0, 1.0,
      1.0, 1.0, 1.0, 1.0, 1.0, 1.0, 1.0, 1.0, 1.0, 1.0, 1.0, 1.0, 1.0, 1.0, 1.0,
      1.0, 1.0, 1.0, 1.0, 1.0, 1.0, 1.0, 1.0, 1.0, 1.0, 1.0, 1.0, 1.0, 1.0, 1.0,
      1.0, 1.0, 1.0, 1.0, 1.0, 1.0, 1.0, 1.0, 1.0, 1.0, 1.0, 1.0, 1.0, 1.0, 1.0,
      1.0, 1.0, 1.0, 1.0, 1.0, 1.0, 1.0, 1.0, 1.0, 1.0, 1.0, 1.0, 1.0, 1.0, 1.0,
      1.0, 1.0, 1.0, 1.0, 1.0, 0.0, 0.0, 0.0, 0.0, 0.0, 0.0, 0.0, 0.0, 0.0, 0.0,
      0.0, 0.0, 0.0, 0.0, 0.0, 0.0, 0.0, 0.0, 0.0, 0.0, 0.0, 0.0, 0.0, 0.0, 0.0,
      1.0, 1.0, 1.0, 1.0, 1.0, 1.0, 1.0, 1.0, 1.0, 1.0, 1.0, 1.0, 1.0, 1.0, 1.0,
      1.0, 1.0, 1.0, 1.0, 1.0, 1.0, 1.0, 1.0, 1.0, 1.0, 1.0, 1.0, 1.0, 1.0, 1.0,
      1.0, 1.0, 1.0, 1.0, 1.0, 1.0, 1.0, 1.0, 1.0, 1.0, 1.0, 1.0, 1.0, 1.0, 1.0,
      1.0, 1.0, 1.0, 1.0, 1.0, 1.0, 1.0, 1.0, 1.0, 1.0, 1.0, 1.0, 1.0, 1.0, 1.0,
      1.0, 1.0, 1.0, 1.0, 1.0, 1.0, 1.0, 1.0, 1.0, 1.0, 1.0, 1.0, 1.0, 1.0, 1.0,
      1.0, 1.0, 1.0, 1.0, 1.0, 1.0, 1.0, 1.0, 0.95000000000000007, -0.05, 0.0,
      0.0, 0.0, 0.0, 0.0, 0.0, 0.0, 0.0, 0.0, 0.0, 0.0, 0.0, 0.0, 0.0, 0.0, 0.0,
      0.0, 0.0, 0.0, 0.0, 0.0, 0.0, 0.0, 0.0, 0.0, 0.0, 0.0, 0.0, 0.0, 0.0, 0.0,
      0.0, 0.0, 0.0, 0.0, 0.0, 0.0, 0.0, 0.0, 0.0, 0.0, 0.0, 0.0, 0.0, 0.0, 0.0,
      0.0, 0.0, 0.0, 0.0, 0.0, 0.0, 0.0, 0.0, 0.0, 0.0, 0.0, 0.0, 0.0, 0.0, 0.0,
      0.0, 0.0, 0.0, 0.0, 0.0, 0.0, 0.0, 0.0, 0.0, 0.0, 0.0, 0.0, 0.0, 0.0, 0.0,
      0.0, 0.0, 0.0, 0.0, 0.0, 0.0, 0.0, 0.0, 0.0, 0.0, 0.0, 0.0, 0.0, 0.0, 0.0,
      0.0, 0.0, 0.0, 0.0, 0.0, 0.0, 0.0, 0.0, 0.0, 0.0, 0.0, 1.0, 1.0, 1.0, 1.0,
      1.0, 0.0, 0.0, 0.0, 0.0, 0.0, 0.0, 0.0, 0.0, 0.0, 0.0, 0.0, 0.0, 0.0, 0.0,
      0.0, 0.0, 0.0, 0.0, 0.0, 0.0, 0.0, 0.0, 0.0, 0.0, 0.0, 0.0, 0.0, 0.0, 0.0,
      0.0, 0.0, 0.0, 0.0, 0.0, 0.0, 0.0, 0.0, 0.0, 0.0, 0.0, 0.0, 0.0, 0.0, 0.0,
      0.0, 0.0, 0.0, 0.0, 0.0, 0.0, 0.0, 0.0, 0.0, 0.0, 0.0, 0.0, 0.0, 0.0, 0.0,
      0.0, 0.0, 0.0, 0.0, 0.0, 0.0, 0.0, 0.0, 0.0, 0.0, 0.0, 0.0, 0.0, 0.0, 0.0,
      0.0, 0.0, 0.0, 0.0, 0.0, 0.0, 0.0, 0.0, 0.0, 0.0, 0.0, 0.0, 0.0, 0.0, 0.0,
      0.0, 0.0, 0.0, 0.0, 0.0, 0.0, 0.0, 0.0, 0.0, 0.0, 0.0, 0.0, 0.0, 0.0, 0.0,
      0.0, 0.0, 0.0, 0.0, 0.0, 0.0, 0.0, 0.0, 0.0, 0.0, 0.0, 0.0, 0.0, 0.0, 0.0,
      0.0, 0.0, 0.0, 0.0, 0.0, 0.0, 0.0, 0.0, 0.0, 0.0, 0.0, 0.0, 0.0, 0.0, 0.0,
      0.0, 0.0, 0.0, 0.0, 0.0, 0.0, 0.0, 0.0, 0.0, 0.0, 0.0, 0.0, 0.0, 0.0, 0.0,
      0.0, 0.0, 0.0, 0.0, 0.0, 0.0, 0.0, 0.0, 0.0, 0.0, 0.0, 0.0, 0.0, 0.0, 0.0,
      0.0, 0.0, 0.0, 0.0, 0.0, 0.0, 0.0, 0.0, 0.0, 0.0, 0.0, 0.0, 0.0, 0.0, 0.0,
      0.0, 0.0, 0.0, 0.0, 0.0, 0.0, 0.0, 0.0, 0.0, 0.0, 0.0, 0.0, 0.0, 0.0, 0.0,
      0.0, 0.0, 0.0, 0.0, 0.0, 0.0, 0.0, 0.0, 0.0, 0.0, 0.0, 0.0, 0.0 } ;

    sltestCruiseControlDefect_DWork.FromWs_PWORK.TimePtr = (void *) pTimeValues0;
    sltestCruiseControlDefect_DWork.FromWs_PWORK.DataPtr = (void *) pDataValues0;
    sltestCruiseControlDefect_DWork.FromWs_IWORK.PrevIndex = 0;
  }

  /* InitializeConditions for UnitDelay: '<S1>/Unit Delay' */
  sltestCruiseControlDefect_DWork.UnitDelay_DSTATE =
    sltestCruiseControlDefective_P.UnitDelay_InitialCondition;

  /* InitializeConditions for UnitDelay: '<S1>/Unit Delay1' */
  sltestCruiseControlDefect_DWork.UnitDelay1_DSTATE =
    sltestCruiseControlDefective_P.UnitDelay1_InitialCondition;

  /* SystemInitialize for Enabled SubSystem: '<S1>/PI Controller' */
  /* InitializeConditions for DiscreteIntegrator: '<S5>/Discrete-Time Integrator' */
  sltestCruiseControlDefect_DWork.DiscreteTimeIntegrator_DSTATE =
    sltestCruiseControlDefective_P.DiscreteTimeIntegrator_IC;

  /* SystemInitialize for Outport: '<Root>/throt' incorporates:
   *  Outport: '<S5>/throt'
   */
  sltestCruiseControlDefective_Y.throt = sltestCruiseControlDefective_P.throt_Y0;

  /* End of SystemInitialize for SubSystem: '<S1>/PI Controller' */
}

/* Model terminate function */
void sltestCruiseControlDefective_terminate(void)
{
  /* (no terminate code required) */
}

/*======================== TOOL VERSION INFORMATION ==========================*
 * MATLAB 9.7 (R2019b)18-Jul-2019                                             *
 * Simulink 10.0 (R2019b)18-Jul-2019                                          *
 * Simulink Coder 9.2 (R2019b)18-Jul-2019                                     *
 * Embedded Coder 7.3 (R2019b)18-Jul-2019                                     *
 * Stateflow 10.1 (R2019b)18-Jul-2019                                         *
 * Fixed-Point Designer 6.4 (R2019b)18-Jul-2019                               *
 *============================================================================*/

/*======================= LICENSE IN USE INFORMATION =========================*
 * matlab                                                                     *
 * matlab_coder                                                               *
 * real-time_workshop                                                         *
 * rtw_embedded_coder                                                         *
 * simulink                                                                   *
 * simulink_test                                                              *
 * stateflow                                                                  *
 *============================================================================*/
```
